{attribute 'linkalways'} 
{attribute 'no_explicit_call' := 'This FB is a CLASS and must be accessed using methods or properties'}
{attribute 'enable_dynamic_creation'}
FUNCTION_BLOCK Node_F_VN_SubtractImageFromScalar EXTENDS VisionNode
VAR
    fScalar : _LREAL(0.0);
    ipSrcImage : _ITcVnImage;
    ipDestImage : _ITcVnImage;
    hrPrev : _HRESULT(S_OK);
	hresult : _HRESULT(S_OK);
END_VAR

METHOD PUBLIC  Clone : I_Node
VAR
	pNode : POINTER TO Node_F_VN_SubtractImageFromScalar;
END_VAR
pNode := __NEW(Node_F_VN_SubtractImageFromScalar);
Clone := pNode^;
END_METHOD

METHOD FB_init : BOOL
VAR_INPUT
	bInitRetains : BOOL; // if TRUE, the retain variables are initialized (warm start / cold start)
	bInCopyCode : BOOL;  // if TRUE, the instance afterwards gets moved into the copy code (online change)
END_VAR
AddInput('fScalar', fScalar);
AddInput('ipSrcImage', ipSrcImage);
AddInput('hrPrev', hrPrev);
AddOutput('ipDestImage', ipDestImage);
AddOutput('hresult',hresult);
END_METHOD

METHOD PROTECTED OnExecute : HRESULT
hresult.Value := F_VN_SubtractImageFromScalar(
    fScalar := fScalar.Value,
    ipSrcImage := ipSrcImage.Value,
	ipDestImage := ipDestImage.Value,
	hrPrev:= hrPrev.Value);
END_METHOD

METHOD PUBLIC PreExecutionCheck
VAR_INPUT
	Check : I_PreExecutionChecks;
END_VAR
IF FAILED(hrPrev.Value) THEN
    RETURN;
END_IF

Check.IsTrue(ipSrcImage.IsValid, 'ipSrcImage must contain an image');
END_METHOD

END_FUNCTION_BLOCK

(* stored: Version 1.1.0.1, ProductVersion 3.1.4024.13
   POU Node_F_VN_SubtractImageFromScalar: Id {8b0808a7-8e3b-0391-37e2-505cab21ffad}, SpecialFunc None
   Folder Constructor: Id {7dcc836e-a4aa-014e-37ab-1ed3e7a4d09e}
   Method Clone: Id {6677bcbc-771f-01ad-3fe6-a414487e7999}
   Method FB_init: Id {c129346e-387c-0db2-1635-9fe8678781cb}
   Method OnExecute: Id {28d0c863-3498-0f5e-135d-cd0d20605839}
   Method PreExecutionCheck: Id {27ad8559-ce55-0c7b-27b6-af363de7eaba} *)
